Fanuc KAREL source: IO0058.KL

-- PROVISIONAL review KL for V1013-1; original PC SHA256 cfdac4b48b9be927cc3c0471e79c59767be705bde3b81b03a6c1b797094a0e2d
-- Incomplete behavior may be omitted. Consult companion uncertainty JSON. Do not deploy.
PROGRAM IO0058
%NOLOCKGROUP
-- UNRESOLVED_LOCAL_POOL 5 cells at code offset 13; source declarations unknown
-- DIRECT_LOCAL_WORD_ACCESS alone does not prove INTEGER, REAL, or BOOLEAN
BEGIN
  -- UNRESOLVED_PC offsets 0-18; opcodes 2B,2C,7B
  -- UNRESOLVED_PC offsets 23-30; opcodes 9D,23
  -- UNRESOLVED_PC offsets 35-49; opcodes 2E,22,9D,33,35
  -- UNRESOLVED_PC offsets 54-61; opcodes 9D,23
  -- UNRESOLVED_PC offsets 66-77; opcodes 2E,23
  -- UNRESOLVED_PC offsets 82-98; opcodes 21,9D,52,19,23
  -- UNRESOLVED_PC offsets 103-107; opcodes 7F
  -- UNRESOLVED_PC offsets 112-116; opcodes 27,AA
  -- UNRESOLVED_PC offsets 121-125; opcodes 7F
END IO0058
